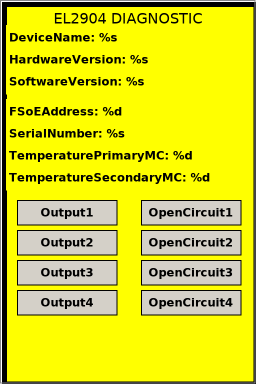
VISUALIZATION V_PH_EL2904_DIAG  // 256x384
VAR_INPUT
	stEL2904DiagnosticData		:ST_EL2904_DiagnosticData;
END_VAR
    Rectangle (2,2 256x384), colour toggle: stEL2904DiagnosticData.bGeneralError
    Label (5,6 246x25), "EL2904 DIAGNOSTIC"
    Rectangle (6,25 242x25), "DeviceName: %s", text variable: stEL2904DiagnosticData.sDeviceName
    Rectangle (6,47 242x25), "HardwareVersion: %s", text variable: stEL2904DiagnosticData.sHardwareVersion
    Rectangle (6,69 242x25), "SoftwareVersion: %s", text variable: stEL2904DiagnosticData.sSoftwareVersion
    Rectangle (6,99 242x25), "FSoEAddress: %d", text variable: stEL2904DiagnosticData.dwFSoEAddress
    Rectangle (6,121 242x25), "SerialNumber: %s", text variable: stEL2904DiagnosticData.sSerialNumber
    Rectangle (6,143 242x25), "TemperaturePrimaryMC: %d", text variable: stEL2904DiagnosticData.wTemperaturePrimaryMC
    Rectangle (6,165 242x25), "TemperatureSecondaryMC: %d", text variable: stEL2904DiagnosticData.wTemperatureSecondaryMC
    RoundedRectangle (17,200 100x25), "Output1", colour toggle: stEL2904DiagnosticData.bOutput1
    RoundedRectangle (17,230 100x25), "Output2", colour toggle: stEL2904DiagnosticData.bOutput2
    RoundedRectangle (17,260 100x25), "Output3", colour toggle: stEL2904DiagnosticData.bOutput3
    RoundedRectangle (17,290 100x25), "Output4", colour toggle: stEL2904DiagnosticData.bOutput4
    RoundedRectangle (141,200 100x25), "OpenCircuit1", colour toggle: stEL2904DiagnosticData.bOutputOpen1, invisible if: NOT stEL2904DiagnosticData.bOutputOpen1
    RoundedRectangle (141,230 100x25), "OpenCircuit2", colour toggle: stEL2904DiagnosticData.bOutputOpen2, invisible if: NOT stEL2904DiagnosticData.bOutputOpen2
    RoundedRectangle (141,260 100x25), "OpenCircuit3", colour toggle: stEL2904DiagnosticData.bOutputOpen3, invisible if: NOT stEL2904DiagnosticData.bOutputOpen3
    RoundedRectangle (141,290 100x25), "OpenCircuit4", colour toggle: stEL2904DiagnosticData.bOutputOpen4, invisible if: NOT stEL2904DiagnosticData.bOutputOpen4
END_VISUALIZATION

(* stored: Version 1.1.0.1, ProductVersion 3.1.4024.4
   Visu V_PH_EL2904_DIAG: Id {a88aa2a5-9c43-4c58-b9ac-9abfb1cb4df0} *)
